FUNCTION_BLOCK ioControl
VAR_INPUT
END_VAR
VAR_OUTPUT
END_VAR
VAR
END_VAR


// Този блок има няколко метода който помагат за по-лесна работа на стъпковата машина
// 1. Метод за преминаване от състояние в състояние
// 2. Конфигурация на самата стъпкова машина
// 3. Няколко метода за четене и завпис на IO сигнали
// 4. State Taimer на базата на който да се генерира аларма

METHOD getSR : BOOL
VAR_INPUT

	xOn:  imageIO;      // Сигнал който трябва да е ON
    XOff: imageIO;      // Сигла който трябва да е OFF	

END_VAR

// Резултата се връща когато единият сигнал е ON, a другият ОFF
// Основно при друпозиционни устр.

IF getX(xOn) AND NOT getX(xOff) THEN
	getSR := TRUE;
ELSE
	getSR := FALSE;	
END_IF
END_METHOD

METHOD getX : BOOL

VAR_INPUT
	
		x	   : imageIO; 		// IO поле
		
END_VAR

VAR
	
		tempByte  : BYTE;
		mask      : BYTE;
		res       : BYTE;
		
END_VAR

// Прочита даден IO сигнал 

IF x.iType = ioType.INPUT_BIT THEN

	IF NOT DEBUG.ioDebugActive THEN	

		tempByte 		 := x.image^[x.iByte];       // Взима байта от IO Image
		mask     		 := SHL(1, x.iBit);         // Подготвя маската
  	 	 res              := tempByte AND mask;
		IF (res = 0) THEN
			getX   := FALSE;
			x.stIO := FALSE; 
		ELSE
			getX   := TRUE;
			x.stIO := TRUE; 
		END_IF
	ELSE	
		IF x.stIO THEN
			getX := TRUE;
		ELSE
			getX := FALSE;
		END_IF
	
	END_IF
	
END_IF
END_METHOD

METHOD rstY
VAR_INPUT
	
	y		: imageIO; 		// поле с IO изходен сигнал

END_VAR

VAR 
	  
	tempByte  : BYTE;
	mask      : BYTE;       // маска за сетване на опредене бит от байта
	
END_VAR
 // Ресетва изходен сигнал в периферията и в Station IO

 IF y.iType = ioType.OUTPUT_BIT THEN
	 
	IF NOT DEBUG.ioDebugActive THEN
	 
		y.stIO   		 := FALSE;         			//  Задава стойността в Station IO

		tempByte 		 := y.image^[y.iByte];       // Взима байта от IO Image
		mask     		 := SHL(1, y.iBit);         // Подготвя маската
		mask             := NOT mask; 				// Инвертирая
		y.image^[y.iByte] := tempByte AND mask;      // Ресетване на желаният бит
		
	ELSE
		y.stIO   		 := FALSE;         			//  Задава стойността в Station IO
END_IF
	
END_IF
END_METHOD

METHOD setSR
VAR_INPUT
	
	yOn:  imageIO;      // Изход който трябва да се сетне
    yOff: imageIO;      // Изход който трябва да се ресетне	

END_VAR

// Сетва първия и ресетва втория сигнал 
// За цилиндри основно

setY(yOn);
rstY(yOff);
END_METHOD

METHOD setY
VAR_INPUT
	
	y		: imageIO; 		// поле с IO изходен сигнал

END_VAR

VAR 
	  
	tempByte  : BYTE;
	mask      : BYTE;       // маска за сетване на опредене бит от байта
	
END_VAR

// Сетва изходен сигнал в периферията и в Station IO

IF y.iType = ioType.OUTPUT_BIT THEN
	
	IF NOT DEBUG.ioDebugActive THEN

		y.stIO           := TRUE;         			//  Задава стойността в Station IO
	
		tempByte 		 := y.image^[y.iByte];       // Взима байта от IO Image
		mask     		 := SHL(1, y.iBit);         // Подготвя маската
		y.image^[y.iByte] := tempByte OR mask;       // Сетване на желаният бит
		
	ELSE
		y.stIO           := TRUE;         			//  Задава стойността в Station IO
END_IF
	
END_IF
END_METHOD

END_FUNCTION_BLOCK

(* stored: Version 1.1.0.1, ProductVersion 3.1.4024.3
   POU ioControl: Id {045ac296-4cd6-48ab-b1e4-b4c57de1a0b8}, SpecialFunc None
   Method getSR: Id {115e0f62-28bd-4ce6-b217-e508967feb4c}
   Method getX: Id {74f1d238-8bc5-48a2-91e8-a504e608b903}
   Method rstY: Id {ad0d7e10-2bf5-40c0-8317-1fa0931fa315}
   Method setSR: Id {f0c1418b-ecec-4c47-a3b6-2e0ad3ddde83}
   Method setY: Id {1e0eccc8-1a2f-4bfd-84dc-bf38688e25f5} *)
